FUNCTION_BLOCK PRINT_TOOL_CHANGE_DATA (* Prints on the terminal the tool to change *)
  (* Standard: 61499-2 *)
  (* Version 1.0, 18-04-2012, GASR, Universidade do Estado de Santa Catarina *)
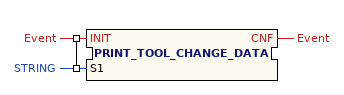
  EVENT_INPUT
    INIT WITH S1;
  END_EVENT
  EVENT_OUTPUT
    CNF;
  END_EVENT
  VAR_INPUT
    S1 : STRING; (* String 1 *)
  END_VAR
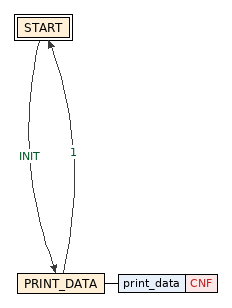
  EC_STATES
    START;
    PRINT_DATA : print_data -> CNF;
  END_STATES
  EC_TRANSITIONS
    START TO PRINT_DATA := INIT;
    PRINT_DATA TO START := 1;
  END_TRANSITIONS
  ALGORITHM print_data IN Lua:
print( "Change tool for"..S1 )
  END_ALGORITHM
END_FUNCTION_BLOCK
